// TIA Portal V18 export
TYPE "PLCtoMES_PrintExchange"
// stored: IsFailsafeCompliant false
   STRUCT
      "P-PrintReq" : Bool;   // 打刻请求
      "P-PrintPartID" : Array[1..10] of String[48];   // PLC请求MES打印内容时发送产品序列号（有RFID则从RFID读取，无RFID，从扫码枪获取）
      Reserve : Array[1..498] of Byte;   // PrintData交互预留
   END_STRUCT;
END_TYPE
